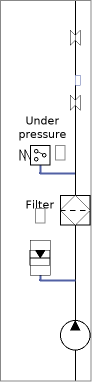
VISUALIZATION VISU_HydraulicsFigure_Pipe  // 92x382
VAR_IN_OUT
	underpressureOK : BOOL;
    filterOK : BOOL;
END_VAR
    Line (75,0) (75,75)
    Polyline (40,165) (40,173) (75,173)
    Line (75,215) (75,320)
    Ellipse (60,320 30x30)
    Polygon (70,330) (75,320) (80,330)
    Line (75,350) (75,380)
    Rectangle (60,195 30x30)
    Polygon (60,210) (75,195) (90,210) (75,225)
    Line (60,210) (65,210)
    Line (80,210) (85,210)
    Line (70,210) (75,210)
    Line (75,85) (75,195)
    Polygon (75,75) (80,75) (80,85) (75,85)
    Rectangle (30,145 20x20)
    Polyline (20,160) (20,150) (25,160) (25,150) (30,160)
    Line (35,150) (45,155)
    Ellipse (34,149 4x4)
    Ellipse (34,157 4x4)
    Ellipse (42,153 4x4)
    Label (10,110 65x35), "Under pressure"
    Label (20,195 40x20), "Filter"
    Frame (55,145 10x15)
        shows VISU_State_red_green(state := underpressureOK)
    Frame (35,208 10x15)
        shows VISU_State_red_green(state := filterOK)
    Polygon (30,250) (30,240) (50,240) (50,250)
    Line (50,265) (50,250)
    Line (30,265) (30,250)
    Line (50,258) (30,258)
    Polygon (35,250) (40,258) (45,250)
    Polyline (40,272) (40,280) (75,280)
    Polygon (30,265) (30,275) (50,275) (50,265)
    Polygon (70,95) (75,100) (75,105) (70,110)
    Polygon (80,95) (75,100) (75,105) (80,110)
    Polygon (70,30) (75,35) (75,40) (70,45)
    Polygon (80,30) (75,35) (75,40) (80,45)
END_VISUALIZATION

(* stored: Version 1.1.0.1, ProductVersion 3.1.4019.2
   Visu VISU_HydraulicsFigure_Pipe: Id {b53e4ea8-fe45-48ff-89d8-6e9ebd846bf0} *)
